SYSTEM TEST_MATRIX (* Test IN_MATRIX with OUT_MATRIX *)
  (* Standard: 61499-1 *)
  (* Version 0.4, 2007-12-26, JHC, Holobloc Inc, Added use of OUT_QO_US. *)
  (* Version 0.4, 2007-12-17, JHC, Holobloc Inc, Added QO, STATUS outputs + labels. *)
  (* Version 0.3, 2007-11-10, JHC, Holobloc Inc, Added tests of all functions. *)
  (* Version 0.2, 2007-05-11, JHC, Holobloc Inc, Updated to new MATRIX, IN_MATRIX, OUT_MATRIX implementations. *)
  (* Version 0.1, 2007-03-15, JHC, Holobloc Inc, Updated to new MATRIX, IN_MATRIX, OUT_MATRIX implementations. *)
  (* Version 0.0, 2004-06-20, JHC, Rockwell Automation *)
  DEVICE MATRIX_TEST : FRAME_DEVICE(BOUNDS := [100,100,470,440], GRID := [4,2])
    RESOURCE IN1 : PANEL_RESOURCE
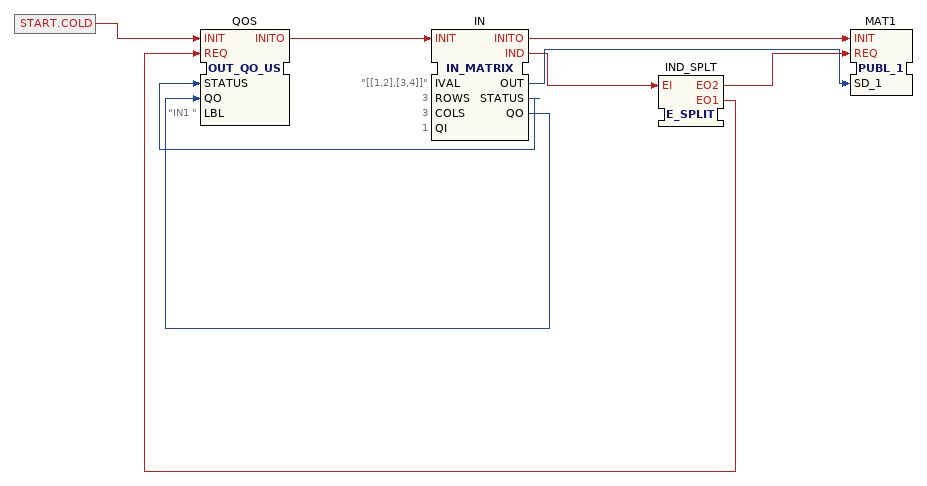
      FBS
        IN : IN_MATRIX(IVAL := "[[1,2],[3,4]]", ROWS := 3, COLS := 3, QI := 1);
        MAT1 : PUBL_1;
        QOS : OUT_QO_US(LBL := "IN1  ");
        IND_SPLT : E_SPLIT;
      END_FBS
      EVENT_CONNECTIONS
        IN.INITO TO MAT1.INIT;
        START.COLD TO QOS.INIT;
        QOS.INITO TO IN.INIT;
        IN.IND TO IND_SPLT.EI;
        IND_SPLT.EO2 TO MAT1.REQ;
        IND_SPLT.EO1 TO QOS.REQ;
      END_CONNECTIONS
      DATA_CONNECTIONS
        IN.OUT TO MAT1.SD_1;
        IN.STATUS TO QOS.STATUS;
        IN.QO TO QOS.QO;
      END_CONNECTIONS
    END_RESOURCE
    RESOURCE IN2 : PANEL_RESOURCE
      FBS
        IN : IN_MATRIX(IVAL := "[[1,2],[3,4],[5,6,7]]", ROWS := 3, COLS := 3, QI := 1);
        MAT2 : PUBL_1;
        QOS : OUT_QO_US(LBL := "IN2  ");
        IND_SPLT : E_SPLIT;
      END_FBS
      EVENT_CONNECTIONS
        IN.INITO TO MAT2.INIT;
        START.COLD TO QOS.INIT;
        QOS.INITO TO IN.INIT;
        IN.IND TO IND_SPLT.EI;
        IND_SPLT.EO2 TO MAT2.REQ;
        IND_SPLT.EO1 TO QOS.REQ;
      END_CONNECTIONS
      DATA_CONNECTIONS
        IN.OUT TO MAT2.SD_1;
        IN.STATUS TO QOS.STATUS;
        IN.QO TO QOS.QO;
      END_CONNECTIONS
    END_RESOURCE
    RESOURCE TEST_OUT : PANEL_RESOURCE
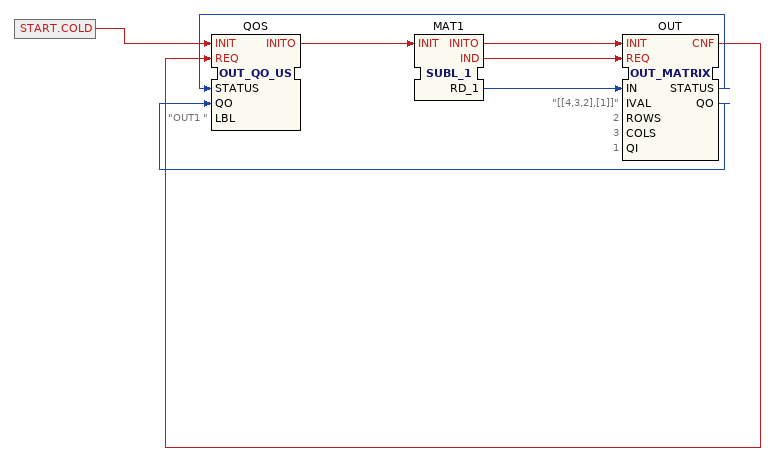
      FBS
        OUT : OUT_MATRIX(IVAL := "[[4,3,2],[1]]", ROWS := 2, COLS := 3, QI := 1);
        MAT1 : SUBL_1;
        QOS : OUT_QO_US(LBL := "OUT1  ");
      END_FBS
      EVENT_CONNECTIONS
        MAT1.INITO TO OUT.INIT;
        MAT1.IND TO OUT.REQ;
        START.COLD TO QOS.INIT;
        QOS.INITO TO MAT1.INIT;
        OUT.CNF TO QOS.REQ;
      END_CONNECTIONS
      DATA_CONNECTIONS
        MAT1.RD_1 TO OUT.IN;
        OUT.STATUS TO QOS.STATUS;
        OUT.QO TO QOS.QO;
      END_CONNECTIONS
    END_RESOURCE
    RESOURCE TEST_ADD : PANEL_RESOURCE
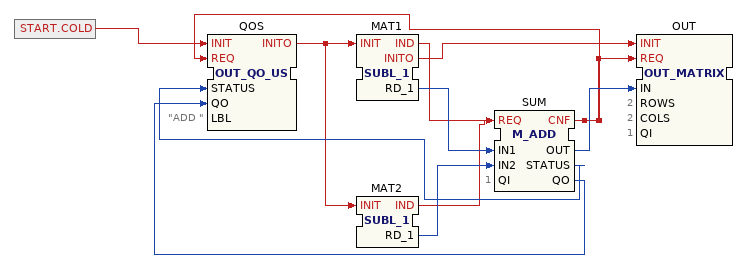
      FBS
        MAT1 : SUBL_1;
        MAT2 : SUBL_1;
        SUM : M_ADD(QI := 1);
        OUT : OUT_MATRIX(ROWS := 2, COLS := 2, QI := 1);
        QOS : OUT_QO_US(LBL := "ADD  ");
      END_FBS
      EVENT_CONNECTIONS
        MAT1.IND TO SUM.REQ;
        MAT1.INITO TO OUT.INIT;
        MAT2.IND TO SUM.REQ;
        SUM.CNF TO OUT.REQ;
        START.COLD TO QOS.INIT;
        QOS.INITO TO MAT1.INIT;
        QOS.INITO TO MAT2.INIT;
        SUM.CNF TO QOS.REQ;
      END_CONNECTIONS
      DATA_CONNECTIONS
        MAT1.RD_1 TO SUM.IN1;
        MAT2.RD_1 TO SUM.IN2;
        SUM.OUT TO OUT.IN;
        SUM.STATUS TO QOS.STATUS;
        SUM.QO TO QOS.QO;
      END_CONNECTIONS
    END_RESOURCE
    RESOURCE TEST_SUB : PANEL_RESOURCE
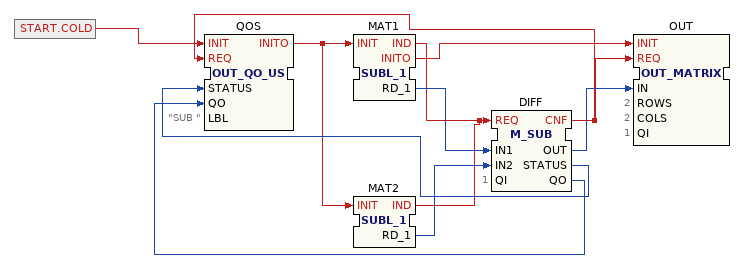
      FBS
        MAT1 : SUBL_1;
        MAT2 : SUBL_1;
        DIFF : M_SUB(QI := 1);
        OUT : OUT_MATRIX(ROWS := 2, COLS := 2, QI := 1);
        QOS : OUT_QO_US(LBL := "SUB  ");
      END_FBS
      EVENT_CONNECTIONS
        MAT1.IND TO DIFF.REQ;
        MAT1.INITO TO OUT.INIT;
        MAT2.IND TO DIFF.REQ;
        DIFF.CNF TO OUT.REQ;
        START.COLD TO QOS.INIT;
        QOS.INITO TO MAT1.INIT;
        QOS.INITO TO MAT2.INIT;
        DIFF.CNF TO QOS.REQ;
      END_CONNECTIONS
      DATA_CONNECTIONS
        MAT1.RD_1 TO DIFF.IN1;
        MAT2.RD_1 TO DIFF.IN2;
        DIFF.OUT TO OUT.IN;
        DIFF.STATUS TO QOS.STATUS;
        DIFF.QO TO QOS.QO;
      END_CONNECTIONS
    END_RESOURCE
    RESOURCE TEST_MUL : PANEL_RESOURCE
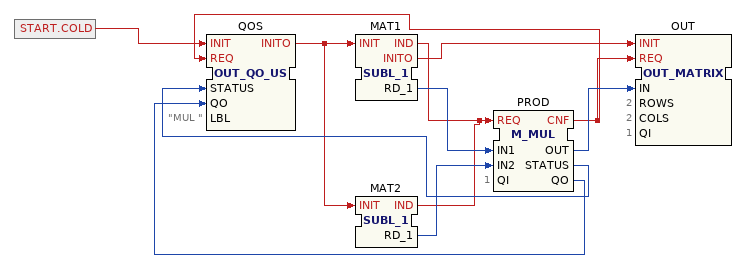
      FBS
        MAT1 : SUBL_1;
        MAT2 : SUBL_1;
        PROD : M_MUL(QI := 1);
        OUT : OUT_MATRIX(ROWS := 2, COLS := 2, QI := 1);
        QOS : OUT_QO_US(LBL := "MUL  ");
      END_FBS
      EVENT_CONNECTIONS
        MAT1.IND TO PROD.REQ;
        MAT1.INITO TO OUT.INIT;
        MAT2.IND TO PROD.REQ;
        PROD.CNF TO OUT.REQ;
        START.COLD TO QOS.INIT;
        QOS.INITO TO MAT1.INIT;
        QOS.INITO TO MAT2.INIT;
        PROD.CNF TO QOS.REQ;
      END_CONNECTIONS
      DATA_CONNECTIONS
        MAT1.RD_1 TO PROD.IN1;
        MAT2.RD_1 TO PROD.IN2;
        PROD.OUT TO OUT.IN;
        PROD.STATUS TO QOS.STATUS;
        PROD.QO TO QOS.QO;
      END_CONNECTIONS
    END_RESOURCE
    RESOURCE TEST_INV : PANEL_RESOURCE
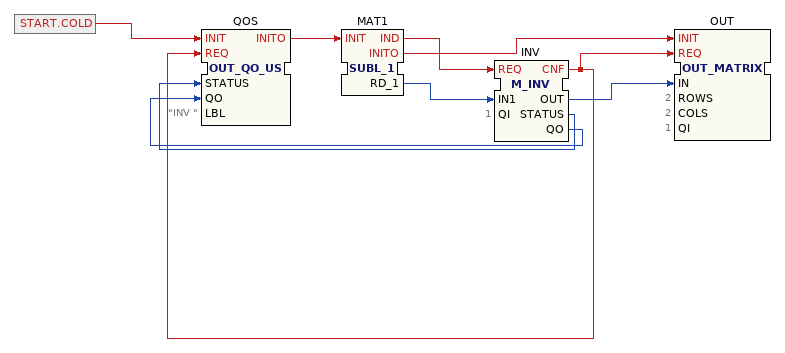
      FBS
        MAT1 : SUBL_1;
        INV : M_INV(QI := 1);
        OUT : OUT_MATRIX(ROWS := 2, COLS := 2, QI := 1);
        QOS : OUT_QO_US(LBL := "INV  ");
      END_FBS
      EVENT_CONNECTIONS
        MAT1.IND TO INV.REQ;
        MAT1.INITO TO OUT.INIT;
        INV.CNF TO OUT.REQ;
        START.COLD TO QOS.INIT;
        QOS.INITO TO MAT1.INIT;
        INV.CNF TO QOS.REQ;
      END_CONNECTIONS
      DATA_CONNECTIONS
        MAT1.RD_1 TO INV.IN1;
        INV.OUT TO OUT.IN;
        INV.STATUS TO QOS.STATUS;
        INV.QO TO QOS.QO;
      END_CONNECTIONS
    END_RESOURCE
  END_DEVICE
END_SYSTEM
